(* CODESYS project copy.project

Project tree, tasks and I/O mapping:
  Device : CODESYS Control Win V3, 3S - Smart Software Solutions GmbH, order no. 305021, version 3.5.9.50
    application Application
      libraries: Standard, * (System); CAA File, 3.5.9.0 (CAA Technical Workgroup); CAA Types Extern, 3.5.5.0 (CAA Technical Workgroup)
      task MainTask (cyclic, interval t#20ms, priority 1) calls PLC_PRG
      program PLC_PRG [ST]
      FileTransfer/
        function block fileTransfer [ST]: start, createDestDir, openDIr, listDir, copyFile, removeFile, closeDir
        data type TransferStatus
        data type TransferError
*)

// Device/Application/FileTransfer/TransferStatus
{attribute 'qualified_only'}
{attribute 'strict'}
TYPE TransferStatus :
(
	iddle := 0,
	createDestDir,
	openDir,
	listDir,
	copyFile,
	removeFile,
	sucess,
	fail,
	closeDir

);
END_TYPE

// Device/Application/FileTransfer/TransferError
{attribute 'qualified_only'}
{attribute 'strict'}
TYPE TransferError :
(
	ok := 0,
	createDestDirError,
	openDirError,
	listDirError,
	copyFileError,
	removeFileError,
	closeDirError
);
END_TYPE

// Device/Application/PLC_PRG
PROGRAM PLC_PRG
VAR
	init:BOOL:=true;
	ft:FileTransfer;
END_VAR




ft();


IF init THEN
	ft.start(
		isSourceDir:='/source/',
		isDestDir:='/dest/ANDERSON/a/',
		ixRemoveFiles:=TRUE,
		iprefixDestFiles:=''
	);	
	init:=FALSE;
END_IF

END_PROGRAM

// Device/Application/FileTransfer/fileTransfer
FUNCTION_BLOCK FileTransfer

VAR_OUTPUT
	xDone:	 	  		BOOL := FALSE;
	xError:				BOOL := FALSE;
END_VAR
VAR   
	sSourceDir:			STRING;
    sDestDir: 			STRING;	
	xRemoveFiles:   	BOOL := FALSE;
	prefixDestFiles:	STRING; 
    Status:         TransferStatus;
    hDir:           CAA.HANDLE;
    deNewDirectory: FILE.FILE_DIR_ENTRY;
    fildcr:         FILE.DirCreate;
    fildop:         FILE.DirOpen;
    fildcl:         FILE.DirClose;
    fildls:         FILE.DirList;
	filcp:  	    FILE.Copy;
	fildl:			FILE.Delete;
	totalSize:  	ULINT;
	tranferSize:  	ULINT;
	wstotalSize:	WSTRING;   
	errorCode:      TransferError; 
	newFileName: CAA.FILENAME;
	
END_VAR

CASE Status OF
	
	TransferStatus.createDestDir: createDestDir();
	TransferStatus.openDir: openDir();	
	TransferStatus.listDir: listDir();
	TransferStatus.copyFile: copyFile();
	TransferStatus.removeFile: removeFile();
	TransferStatus.closeDir: closeDir();	
	TransferStatus.sucess: 
		status:= TransferStatus.closeDir;
		errorCode:= TransferError.ok;
		xDone:=TRUE;
	TransferStatus.fail: 
		status:= TransferStatus.closeDir;
		xError:=TRUE;

END_CASE

METHOD start
VAR_INPUT
    isSourceDir:		STRING;
    isDestDir: 			STRING;	
	ixRemoveFiles:   	BOOL;
	iprefixDestFiles:	STRING; 
END_VAR

sSourceDir:= isSourceDir;		
sDestDir:= isDestDir; 			
xRemoveFiles:= ixRemoveFiles;   
prefixDestFiles:= iprefixDestFiles;

xDone:=FALSE;
xError:=FALSE;

errorCode:= TransferError.ok;

fildcr(xExecute:=FALSE);
fildop(xExecute:=FALSE);
fildcl(xExecute:=FALSE);
fildls(xExecute:=FALSE);	
filcp (xExecute:=FALSE);
fildl (xExecute:=FALSE);
	
totalSize:=0;

Status:=TransferStatus.createDestDir;
END_METHOD

METHOD createDestDir
fildcr.sDirName:=sDestDir;
fildcr.xParent:=TRUE;
IF NOT fildcr.xBusy THEN
	fildcr(xExecute:=TRUE);	
END_IF
IF fildcr.xDone OR fildcr.eError = FILE.ERROR.EXIST THEN
	Status:=TransferStatus.openDir;
END_IF
IF fildcr.xError AND fildcr.eError <> FILE.ERROR.EXIST  THEN
	(* error handling*)
	Status:=TransferStatus.Fail;
	errorCode:= TransferError.createDestDirError;
END_IF
fildcr(xExecute:=FALSE);
END_METHOD

METHOD openDIr
VAR_INPUT
END_VAR
fildop.sDirName:=sSourceDir;
IF NOT fildop.xBusy THEN
	fildop(xExecute:=TRUE);	
END_IF
IF fildop.xDone THEN
	hDir := fildop.hDir;
	Status:=TransferStatus.listDir;
END_IF
IF fildop.xError THEN
	(* error handling*)
	Status:=TransferStatus.Fail;
	errorCode:= TransferError.openDirError;
END_IF
fildop(xExecute:=FALSE);
END_METHOD

METHOD listDir
VAR_INPUT
END_VAR
fildls.hDir:=hDir;
IF NOT fildls.xBusy THEN
	fildls( xExecute:=TRUE);
END_IF		
IF fildls.xDone THEN
	deNewDirectory.sEntry 				:=fildls.deDirEntry.sEntry;
	deNewDirectory.szSize 				:=fildls.deDirEntry.szSize;
	deNewDirectory.xDirectory 			:=fildls.deDirEntry.xDirectory;
	deNewDirectory.xExclusive			:=fildls.deDirEntry.xExclusive;
	deNewDirectory.dtLastModification   :=fildls.deDirEntry.dtLastModification; 



	IF NOT fildls.deDirEntry.xDirectory THEN
		status:=TransferStatus.copyFile;
		//totalSize:= totalSize+caa.SIZE_TO_ULINT(fildls.deDirEntry.szSize);
		//wstotalSize:=BytesToHumanReadable(totalSize);
	END_IF   
END_IF	

IF fildls.eError = FILE.ERROR.NO_MORE_ENTRIES THEN
	status:=TransferStatus.sucess;
	RETURN;
END_IF 

IF fildls.xError AND fildls.eError <> FILE.ERROR.NO_MORE_ENTRIES THEN
	(* error handling*)
	status:=TransferStatus.fail;
	errorCode:= TransferError.listDirError;
END_IF	
fildls( xExecute:=FALSE);
END_METHOD

METHOD copyFile
VAR_INPUT
END_VAR
filcp.sFileNameSource:= CONCAT(sSourceDir, deNewDirectory.sEntry);
newFileName:= CONCAT(prefixDestFiles, deNewDirectory.sEntry);
filcp.sFileNameDest:= CONCAT(sDestDir, newFileName);
filcp.udiTimeOut:= 1000000;  (* 1s Timeout *)
filcp.xOverWrite:= TRUE;     (* overwrite the existing file *)
IF NOT filcp.xBusy THEN
	filcp( xExecute := TRUE );
END_IF	        
IF filcp.xDone THEN
	tranferSize:= tranferSize + CAA.SIZE_TO_ULINT(filcp.szSize);			
	filcp( xExecute := FALSE );
	IF xRemoveFiles THEN
		Status:= TransferStatus.removeFile;  
	ELSE
		Status:= TransferStatus.listDir; 	
	END_IF
END_IF
IF filcp.xError THEN
	(* error handling*)
	Status:= TransferStatus.fail;
	errorCode:= TransferError.copyFileError;
END_IF
filcp( xExecute := FALSE );
END_METHOD

METHOD removeFile
VAR_INPUT
END_VAR
fildl.sFileName:= CONCAT(sSourceDir, deNewDirectory.sEntry);
IF NOT fildl.xBusy THEN
	fildl( xExecute := TRUE );
END_IF	
fildl( xExecute:=TRUE);
IF fildl.xDone THEN
	status:=TransferStatus.listDir;
END_IF
IF fildl.xError THEN
	(* error handling*)
	status:=TransferStatus.fail;
	errorCode:= TransferError.removeFileError;
END_IF
fildl( xExecute := FALSE );
END_METHOD

METHOD closeDir
VAR_INPUT
END_VAR
IF hDir = 0  THEN
	status:=TransferStatus.iddle;
END_IF 	

IF NOT fildcl.xBusy AND NOT fildcl.xDone THEN
	fildcl.hDir:=hDir;
	
	fildcl( xExecute:=TRUE);	
END_IF	

IF fildcl.xDone THEN
	hDir:=0;
END_IF

IF fildcl.xError THEN
	(* error handling*)
	errorCode:= TransferError.closeDirError;
	hDir:=0;
END_IF	

fildcl( xExecute:=FALSE);
END_METHOD

END_FUNCTION_BLOCK
